// TwinCAT 3 PLC project Robotino_PLC_TEST
// ProgramVersion: 3.1.4022.0
// libraries:
//   Tc2_EtherCAT, * (Beckhoff Automation GmbH)
//   Tc2_Standard, * (Beckhoff Automation GmbH)
//   Tc2_System, * (Beckhoff Automation GmbH)
//   Tc2_Utilities, * (Beckhoff Automation GmbH)
//   Tc3_Module, * (Beckhoff Automation GmbH)
// project tree:
//   DUTs/ EnumState.TcDUT
//   / PlcTask.TcTTO
//   POUs/COE_Auswertung/ SDODaten.TcPOU, SDODatenMotor1.TcPOU, SDODatenMotor2.TcPOU, SDODatenMotor3.TcPOU, SDODatenMotorklemme1.TcPOU, SDODatenMotorklemme2.TcPOU
//   POUs/Motoransteuerung/ MAIN_Motoransteuerung.TcPOU
//   POUs/Motormesswerte/ MAIN_Motormesswerte.TcPOU
//   POUs/Shutdown/ MAIN_Shutdown.TcPOU, Shutdown.TcPOU
//   POUs/UDP/ MAIN_UDP.TcPOU, UDPConnect.TcPOU
// real-time tasks:
//   TASK PlcTask: cycle T#400us, priority 1, ADS port 350
//   TASK IrSensorTask: cycle T#1ms, priority 2, ADS port 351
//   TASK UdpTask: cycle T#2ms, priority 3, ADS port 352
//   TASK SimulinkTask: cycle T#5ms, priority 4, ADS port 353
// I/O:
//   DEVICE Gerät 1 (EtherCAT), AmsNetId 5.49.201.214.2.1
//     Klemme 1 (EK1200) [EK1200-5000 EtherCAT Netzteil (2A E-Bus)]
//       Motorklemme 1 [EL7342 2K. DC-Motor-Endstufe (50V, 3.5A)]
//       Motorklemme 2 [EL7342 2K. DC-Motor-Endstufe (50V, 3.5A)]
//       Digitale Eingänge [EL1008 8K. Dig. Eingang 24V, 3ms]
//       Digitale Ausgänge [EL2004 4K. Dig. Ausgang 24V, 0.5A]
//       Analoge Eingänge (8) [EL3068 8K. Ana. Eingang 0-10V]
//       Analog Eingänge (4) [EL3064 4K.Ana. Eingang 0-10V]
//       Netzklemme (5V) [EL9505 Netzteilklemme 5V]
//       Busendklemme [EL9011 Endklemme]
//   DEVICE UDP Adapter
// variable links:
//   Device 1 (EtherCAT) <-> irSensors/irSensors_Obj
//     Term 1 (EK1200)/Analog Eingänge (4)/AI Standard Channel 1/IR9 <-> Inputs/irInputData[8]
//     Term 1 (EK1200)/Analoge Eingänge (8)/AI Standard Channel {1..8}/IR{1..8} <-> Inputs/irInputData[{0..7}]  (8 links)
//   Robotino_PLC_TEST/Robotino_PLC_TEST Instance <-> Device 1 (EtherCAT)/Term 1 (EK1200)/Digitale Eingänge
//     PlcTask Inputs/MAIN_Motoransteuerung.bumper <-> Channel 2/Bumper
//     PlcTask Inputs/Shutdown.bStart <-> Channel 8/Shutdown
//   Robotino_PLC_TEST/Robotino_PLC_TEST Instance <-> Device 1 (EtherCAT)/Term 1 (EK1200)/Motorklemme 1
//     PlcTask Inputs/MAIN_Motormesswerte.encDataFromMotor2 <-> ENC Status compact Channel 2/Counter value
//     PlcTask Inputs/MAIN_Motormesswerte.encDataFromMotor3 <-> ENC Status compact Channel 1/Counter value
//     PlcTask Outputs/MAIN_Motoransteuerung.enableToMotor2 <-> DCM Control Channel 2/Control/Enable
//     PlcTask Outputs/MAIN_Motoransteuerung.enableToMotor3 <-> DCM Control Channel 1/Control/Enable
//     PlcTask Outputs/MAIN_Motoransteuerung.velocityToMotor2 <-> DCM Velocity Channel 2/Velocity
//     PlcTask Outputs/MAIN_Motoransteuerung.velocityToMotor3 <-> DCM Velocity Channel 1/Velocity
//   Robotino_PLC_TEST/Robotino_PLC_TEST Instance <-> Device 1 (EtherCAT)/Term 1 (EK1200)/Motorklemme 2
//     PlcTask Inputs/MAIN_Motormesswerte.encDataFromMotor1 <-> ENC Status compact Channel 1/Counter value
//     PlcTask Outputs/MAIN_Motoransteuerung.enableToMotor1 <-> DCM Control Channel 1/Control/Enable
//     PlcTask Outputs/MAIN_Motoransteuerung.velocityToMotor1 <-> DCM Velocity Channel 1/Velocity
//   Robotino_PLC_TEST/Robotino_PLC_TEST Instance <-> TcCOM Objects/Object2 (Gewerk3_Simulink_Regler)
//     PlcTask Inputs/MAIN_Motoransteuerung.vThetaCartesianToMotors <-> Output/thetaCartesianToMotors
//     PlcTask Inputs/MAIN_Motoransteuerung.vXCartesianToMotors <-> Output/vXCartesianToMotors
//     PlcTask Inputs/MAIN_Motoransteuerung.vYCartesianToMotors <-> Output/vYCartesianToMotors
//     PlcTask Outputs/MAIN_Motormesswerte.vXCartesianFromMotors <-> Input/u5elements[2]
//     PlcTask Outputs/MAIN_Motormesswerte.vYCartesianFromMotors <-> Input/u5elements[3]
//     PlcTask Outputs/MAIN_Motormesswerte.vthetaCartesianFromMotors <-> Input/u5elements[4]
//     PlcTask Outputs/MAIN_UDP.theta[4] <-> Input/UDP[11]
//     PlcTask Outputs/MAIN_UDP.x[4] <-> Input/UDP[9]
//     PlcTask Outputs/MAIN_UDP.y[4] <-> Input/UDP[10]

CONFIGURATION Robotino_PLC_TEST
    RESOURCE PLC ON TwinCAT3
        TASK PlcTask(INTERVAL := T#400us, PRIORITY := 1);
        PROGRAM MAIN_Motoransteuerung WITH PlcTask : MAIN_Motoransteuerung;
        PROGRAM MAIN_Motormesswerte WITH PlcTask : MAIN_Motormesswerte;
        PROGRAM MAIN_Shutdown WITH PlcTask : MAIN_Shutdown;
        PROGRAM MAIN_UDP WITH PlcTask : MAIN_UDP;
        PROGRAM SDODaten WITH PlcTask : SDODaten;
    END_RESOURCE
END_CONFIGURATION

// ---- DUTs/EnumState.TcDUT
{attribute 'qualified_only'}
{attribute 'strict'}
TYPE EnumState :
(
	init,
	drive,
	reset
);
END_TYPE

// ---- POUs/Motoransteuerung/MAIN_Motoransteuerung.TcPOU
PROGRAM MAIN_Motoransteuerung
VAR	
	//Zustandsautomat
	state:		EnumState:=EnumState.init;
	nextState:	EnumState:=EnumState.init;

	//Achsen Freischalten
	enableMotors: BOOL	:=0;

	//Umgerechnete Werte
	vX:		LREAL:=0;
	vY:		LREAL:=0;
	vTheta:	LREAL:=0;
	v1:		LREAL:=0;
	v2:		LREAL:=0;
	v3:		LREAL:=0;
	//Fahrrichtung Motor
	velocityMotor1 :LREAL:=0;
	velocityMotor2 :LREAL:=0;
	velocityMotor3 :LREAL:=0;
	
	//Skalierung auf MaxGeschwindigkeit Skalierung hängt mit CoE Register 8020:07 8020:08 zusammen !!!
	velocityMax:LREAL:=942.4777961;// Nenndrehzahl U/min CoE Register 8020:07 8020:08 fesgelegt Faktor 16 Wegen Getriebe 1:16
	velocityMotorsTf:LREAL:=0;
	
	// Skalierung auf Ansteuersignale LREAL=>WORD   Skalierung hängt mit CoE Register 8020:07 8020:08 zusammen !!!
	skalPos:LREAL:=34.7668668;//  MaxValue/MaxVelocity   [1/ mm/s]   32767/(942mm/s)   MaxVelocity=D*PI*n/(16*60) //16:1 Getriebeübersetzung  
	skalNeg:LREAL:=34.76792783;//  MaxVelau/MaxVelocity   [1/ mm/s]   32768/(942mm/s)   MaxVelocity=(80mm*PI*3600 U/min)/(16*60sec/min)
	
	//Inputs: CartesianToMotors + Bumper
	vXCartesianToMotors 	AT%I*:LREAL:=0;
	vYCartesianToMotors 	AT%I*:LREAL:=0;
	vThetaCartesianToMotors AT%I*:LREAL:=0;
	bumper	   AT%I*: BOOL:=0;
	
	//Outputs: Motor Values and Enable Signal
	enableToMotor1 AT%Q*:BOOL:=FALSE;
	enableToMotor2 AT%Q*:BOOL:=FALSE;
	enableToMotor3 AT%Q*:BOOL:=FALSE;
	
	velocityToMotor1 AT%Q*:INT:=0;
	velocityToMotor3 AT%Q*:INT:=0;
	velocityToMotor2 AT%Q*:INT:=0;
	
END_VAR

// Konverzierung ToMotors Anfang********************************************************

//	  conversion from positive and / or negative longitudinal, lateral and
//	  rotational velocities(in milimeters per second) to three separate
//	  positive motor velocities(resolution: 1Byte) and their rotation
//    direction
//inputs:  	velocityX  (longitudinal velocity in milimeters per second)
//         	velocityY  (lateral velocity in milimeters per second)
//			vtheta     (rotational velocity in milimeters per second)
//outputs : velocityToMotor1	
//			velocityToMotor2
//			velocityToMotor3
//conversion from longitudinal, lateral & rotational velocity to the
//three separate motor velocities
vX:=vXCartesianToMotors;
vY:=vYCartesianToMotors;
vTheta:=vThetaCartesianToMotors;

v1 := (-vX * COS(30.0*PI/180))	+ (vY * COS(60.0*PI/180))	+ (vTheta * 135.0);
v2 := 0.0						+ (-vY)						+ (vTheta * 135.0);
v3 := (vX * COS(30.0*PI/180))	+ (vY * COS(60.0*PI/180))	+ (vTheta * 135.0);
	
//Drehrichtung Umkehren
velocityMotor1:=-v1;
velocityMotor2:=-v2;
velocityMotor3:=-v3;

//Geschwindigkeitsbegrenzung
IF velocityMotor1 > velocityMax THEN
    velocityMotorsTf:= velocityMotor1;
    
    velocityMotor1:= velocityMax;
    velocityMotor2:= velocityMax * velocityMotor2 / velocityMotorsTf;
    velocityMotor3:= velocityMax * velocityMotor3 / velocityMotorsTf;
END_IF

IF velocityMotor2 > velocityMax THEN
    velocityMotorsTf:= velocityToMotor2;
    
    velocityMotor1:= velocityMax * velocityToMotor1 / velocityMotorsTf;
    velocityMotor2:= velocityMax;
    velocityMotor3:= velocityMax * velocityToMotor3 / velocityMotorsTf;
END_IF

IF velocityMotor3 > velocityMax THEN
    velocityMotorsTf:= velocityToMotor3;
    
    velocityMotor1:= velocityMax * velocityMotor1 / velocityMotorsTf;
    velocityMotor2:= velocityMax * velocityMotor2 / velocityMotorsTf;
    velocityMotor3:= velocityMax;
END_IF
// Konverzierung ToMotors ENDE********************************************************


//MOTORANSTEUERUNG Zustandsautomat

CASE state OF
	EnumState.init:						
						IF bumper=TRUE THEN
							nextState:=EnumState.reset;
							ELSE
								nextState:=EnumState.drive;
						END_IF
	EnumState.drive:
						IF velocityMotor1>=0 THEN
							velocityToMotor1:=LREAL_TO_INT(velocityMotor1*skalPos);
						ELSE
							velocityToMotor1:=LREAL_TO_INT(velocityMotor1*skalNeg);
						END_IF
						
						IF velocityMotor2>=0 THEN
							velocityToMotor2:=LREAL_TO_INT(velocityMotor2*skalPos);
						ELSE
							velocityToMotor2:=LREAL_TO_INT(velocityMotor2*skalNeg);
						END_IF
						
						IF velocityMotor3>=0 THEN
							velocityToMotor3:=LREAL_TO_INT(velocityMotor3*skalPos);
						ELSE
							velocityToMotor3:=LREAL_TO_INT(velocityMotor3*skalNeg); 
						END_IF
							
							enableToMotor1:=1;
							enableToMotor2:=1;
							enableToMotor3:=1;
							
						IF bumper=TRUE THEN
							nextState:=EnumState.reset;
						END_IF
	EnumState.reset:
						velocityToMotor1:=0;
						velocityToMotor2:=0;
						velocityToMotor3:=0;
						enableToMotor1:=0;
						enableToMotor2:=0;
						enableToMotor3:=0;
	ELSE
		nextState:=EnumState.reset;
END_CASE
state:=nextState;

END_PROGRAM

// ---- POUs/Motormesswerte/MAIN_Motormesswerte.TcPOU
PROGRAM MAIN_Motormesswerte
VAR
bStart: BOOL := FALSE;	

//ENC Daten Differenzieren für Geschwindigkeit
diffConst:LREAL:=0.0004;//SECONDS
encDataOldMotor1:UINT:=0;
encDataOldMotor2:UINT:=0;
encDataOldMotor3:UINT:=0;

//Koordinatentransformation Weg
skalEnc:LREAL:=0.00766990393;
x1:LREAL:=0;
x2:LREAL:=0;
x3:LREAL:=0;

xFromMotor1:LREAL:=0;
xFromMotor2:LREAL:=0;
xFromMotor3:LREAL:=0;

//Koordinatentransformation Geschwindigkeit
v1:LREAL:=0;
v2:LREAL:=0;
v3:LREAL:=0;
velocityFromMotor1:LREAL:=0;
velocityFromMotor2:LREAL:=0;
velocityFromMotor3:LREAL:=0;

//INPUTS
encDataFromMotor1 AT%I*  :UINT:=0;
encDataFromMotor2 AT%I*  :UINT:=0;
encDataFromMotor3 AT%I*  :UINT:=0;

diff:  INT :=0;
diff1: INT := 0;
diff2: INT := 0;
diff3: INT := 0;

//OUTPUTS
posXCartesianFromMotors AT%Q*:LREAL:=0;
posYCartesianFromMotors AT%Q*:LREAL:=0;
posThetaCartesianFromMotors AT%Q*:LREAL:=0;

vXCartesianFromMotors AT%Q*:LREAL:=0;
vYCartesianFromMotors AT%Q*:LREAL:=0;
vthetaCartesianFromMotors AT%Q*:LREAL:=0;
END_VAR

IF bStart = FALSE THEN
	encDataOldMotor1 := encDataFromMotor1;
	encDataOldMotor2 := encDataFromMotor2;
	encDataOldMotor3 := encDataFromMotor3;
	bStart := TRUE;
END_IF



// Encoder Wegberechnung und Differenzierung für Geschwindigkeit
diff1:=UINT_TO_INT(encDataFromMotor1) - UINT_TO_INT(encDataOldMotor1);
IF diff1 >= 32767 OR diff1 <= -32767 THEN
	diff1 := 0;
END_IF
diff2:=UINT_TO_INT(encDataFromMotor2) - UINT_TO_INT(encDataOldMotor2);
IF diff2 >= 32767 OR diff2 <= -32767 THEN
	diff2 := 0;
END_IF
diff3:=UINT_TO_INT(encDataFromMotor3) - UINT_TO_INT(encDataOldMotor3);
IF diff3 >= 32767 OR diff3 <= -32767 THEN
	diff3 := 0;
END_IF

xFromMotor1:=xFromMotor1+diff1*skalEnc;
velocityFromMotor1:=diff1/diffConst*skalEnc;

xFromMotor2:=xFromMotor2+diff2*skalEnc;
velocityFromMotor2:=diff2/diffConst*skalEnc;

xFromMotor3:=xFromMotor3+diff3*skalEnc;
velocityFromMotor3:=diff3/diffConst*skalEnc;

// Koordinatentransformation Weg
x1:=-xFromMotor1;
x2:=-xFromMotor2;
x3:=-xFromMotor3;

posXCartesianFromMotors:=(x3 - x1) / (2.0 * COS(30.0*PI/180));  //in mm / s
posYCartesianFromMotors:=(x1 - 2.0 * x2 + x3) / 3.0;            //in mm / s
posThetaCartesianFromMotors:=(x1 + x2 + x3) / (3.0 * 135.0);    //in rad / s

// Koordinatentransformation Geschwindigkeit
v1:=-velocityFromMotor1;
v2:=-velocityFromMotor2;
v3:=-velocityFromMotor3;

vXCartesianFromMotors:=(v3 - v1) / (2.0 * COS(30.0*PI/180));  //in mm / s
vYCartesianFromMotors:=(v1 - 2.0 * v2 + v3) / 3.0;            //in mm / s
vThetaCartesianFromMotors:=(v1 + v2 + v3) / (3.0 * 135.0);    //in rad / s

// Alte Encoderdaten speichern

encDataOldMotor1:=encDataFromMotor1;
encDataOldMotor2:=encDataFromMotor2;
encDataOldMotor3:=encDataFromMotor3;

END_PROGRAM

// ---- POUs/Shutdown/MAIN_Shutdown.TcPOU
PROGRAM MAIN_Shutdown
VAR
END_VAR

Shutdown();

END_PROGRAM

// ---- POUs/Shutdown/Shutdown.TcPOU
PROGRAM Shutdown
VAR
	bStart	AT%I* : BOOL := FALSE;
	Shutdown_Block: NT_Shutdown;
END_VAR

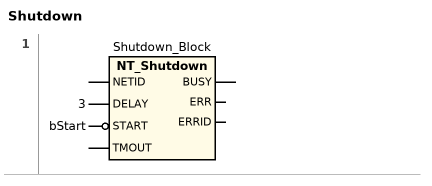
// NETWORK 1
Shutdown_Block(DELAY := 3, START := NOT bStart); // NT_Shutdown

END_PROGRAM

// ---- POUs/UDP/MAIN_UDP.TcPOU
PROGRAM MAIN_UDP
VAR
	//sPaketinhalt	: LREAL;
	//nPaketlaenge	: UDINT;
	
	x	  AT%Q*	: ARRAY[1..4] OF LREAL;
	y	  AT%Q*	: ARRAY[1..4] OF LREAL;
	theta AT%Q*	: ARRAY[1..4] OF LREAL;
	udp1 : UDPConnect;
END_VAR

udp1();

END_PROGRAM

// ---- POUs/UDP/UDPConnect.TcPOU
{attribute 'c++_compatible'}
FUNCTION_BLOCK UDPConnect IMPLEMENTS ITcIoUdpProtocolRecv
VAR_INPUT
END_VAR
VAR_OUTPUT
END_VAR
VAR
	{attribute 'TcInitSymbol'}
    oid:              OTCID; 
    ipUdp:            ITcIoUdpProtocol;
    updPort:          UINT := 25000;
    nReceivedPakets:  UINT;
    hrInit :          HRESULT;
    hrSend :          HRESULT;
END_VAR

IF ipUdp <> 0 THEN
    ipUdp.CheckReceived();
END_IF

METHOD FB_exit : BOOL
VAR_INPUT
	bInCopyCode : BOOL; // if TRUE, the exit method is called for exiting an instance that is copied afterwards (online change).
END_VAR
IF (NOT bInCopyCode AND ipUdp <> 0) THEN //Shutdown
     ipUdp.UnregisterReceiver(updPort);
    FW_SafeRelease(ADR(ipUdp));
     FB_exit := TRUE;
ELSE
     FB_exit := FALSE;
END_IF
END_METHOD

METHOD FB_init : BOOL
VAR_INPUT
	bInitRetains : BOOL; // if TRUE, the retain variables are initialized (warm start / cold start)
	bInCopyCode : BOOL;  // if TRUE, the instance afterwards gets moved into the copy code (online change)
END_VAR

VAR
    ipSrv: ITComObjectServer;
    hr : HRESULT;
END_VAR
IF NOT bInCopyCode THEN // no online change
    IF ipUdp = 0 THEN
     hrInit := FW_ObjMgr_GetObjectInstance(   oid:=oid, 
    
    iid:=TC_GLOBAL_IID_LIST.IID_ITcIoUdpProtocol, 

    pipUnk:=ADR(ipUdp) );
        IF ( SUCCEEDED(hr) AND ipUdp.RegisterReceiver(updPort, THIS^) = 0 ) THEN //open port
            FB_init := TRUE;
        ELSE
            FB_init := FALSE; 
            FW_SafeRelease(ADR(ipUdp));
        END_IF
    END_IF
END_IF
END_METHOD

METHOD FB_reinit : BOOL
VAR_INPUT
END_VAR
IF (ipUdp <> 0) THEN 
 ipUdp.RegisterReceiver(updPort, THIS^);
END_IF
END_METHOD

{attribute 'object_name' := 'ReceiveData'}
{attribute 'c++_compatible'}
{attribute 'signature_flag' := '33554688'}
{attribute 'pack_mode' := '4'}
{attribute 'show'}
{attribute 'minimal_input_size' := '4'}
METHOD ReceiveData : HRESULT
VAR_INPUT
	ipAddr	: UDINT;
	udpDestPort	: UINT;
	udpSrcPort	: UINT;
	nData	: UDINT;
	pData	: PVOID;
	pVlan	: POINTER TO ETYPE_VLAN_HEADER := 0;
END_VAR

VAR
	i	: ULINT := 0;
END_VAR
nReceivedPakets := nReceivedPakets+1;
//MAIN_UDP.nPaketlaenge := nData;

FOR i := 0 TO 3 DO
	memcpy(ADR(MAIN_UDP.x[i+1]),pData+((i*3)*8),8);
	memcpy(ADR(MAIN_UDP.y[i+1]),pData+((i*3+1)*8),8);
	memcpy(ADR(MAIN_UDP.theta[i+1]),pData+((i*3+2)*8),8);
END_FOR;
END_METHOD

{attribute 'c++_compatible'}
{attribute 'minimal_input_size' := '4'}
{attribute 'pack_mode' := '4'}
{warning 'Methodenimplementierung hinzufügen'}
METHOD TcAddRef : UDINT
END_METHOD

{attribute 'c++_compatible'}
{attribute 'minimal_input_size' := '4'}
{attribute 'pack_mode' := '4'}
{warning 'Methodenimplementierung hinzufügen'}
METHOD TcQueryInterface : HRESULT
VAR_INPUT
	iid	: REFERENCE TO IID;
	pipItf	: POINTER TO PVOID;
END_VAR
END_METHOD

{attribute 'c++_compatible'}
{attribute 'minimal_input_size' := '4'}
{attribute 'pack_mode' := '4'}
{warning 'Methodenimplementierung hinzufügen'}
METHOD TcRelease : UDINT
END_METHOD

END_FUNCTION_BLOCK

// ---- POUs/COE_Auswertung/SDODaten.TcPOU
PROGRAM SDODaten
VAR
	DatenMotor1: SDODatenMotor1;
	DatenMotor2: SDODatenMotor2;
	DatenMotor3: SDODatenMotor3;
	DatenMotorklemme1: SDODatenMotorklemme1;
	DatenMotorklemme2: SDODatenMotorklemme2;
END_VAR

DatenMotor1();
DatenMotor2();
DatenMotor3();
DatenMotorklemme1();
DatenMotorklemme2();

END_PROGRAM

// ---- POUs/COE_Auswertung/SDODatenMotor1.TcPOU
FUNCTION_BLOCK SDODatenMotor1
VAR_INPUT
END_VAR
VAR_OUTPUT
	
	Motor1Spannung: UINT;
	Motor1Strom: INT;
	Motor1Strombegrenzung: UINT;
	Motor1Regelfehler: INT;
	Motor1Geschwindigkeit: INT;
	Motor1Overloadtime: UINT;
	Motor1Overtemperature: BOOL;
	Motor1Torqueoverload: BOOL;
	Motor1Shortcirciut: BOOL;
	
END_VAR
VAR
	Motorspannung: FB_EcCoESdoRead;	
	Motorstrom: FB_EcCoESdoRead;
	Strombegrenzung: FB_EcCoESdoRead;
	Regelfehler: FB_EcCoESdoRead;
	Geschwindigkeit: FB_EcCoESdoRead;
	Overload: FB_EcCoESdoRead;
	Short_Circuit: FB_EcCoESdoRead;
	Torque_Overload: FB_EcCoESdoRead;
	Over_Temperature: FB_EcCoESdoRead;

	trigger: BOOL;
	TON_0: TON;
	TON_1: TON;
	ms: TIME;

END_VAR

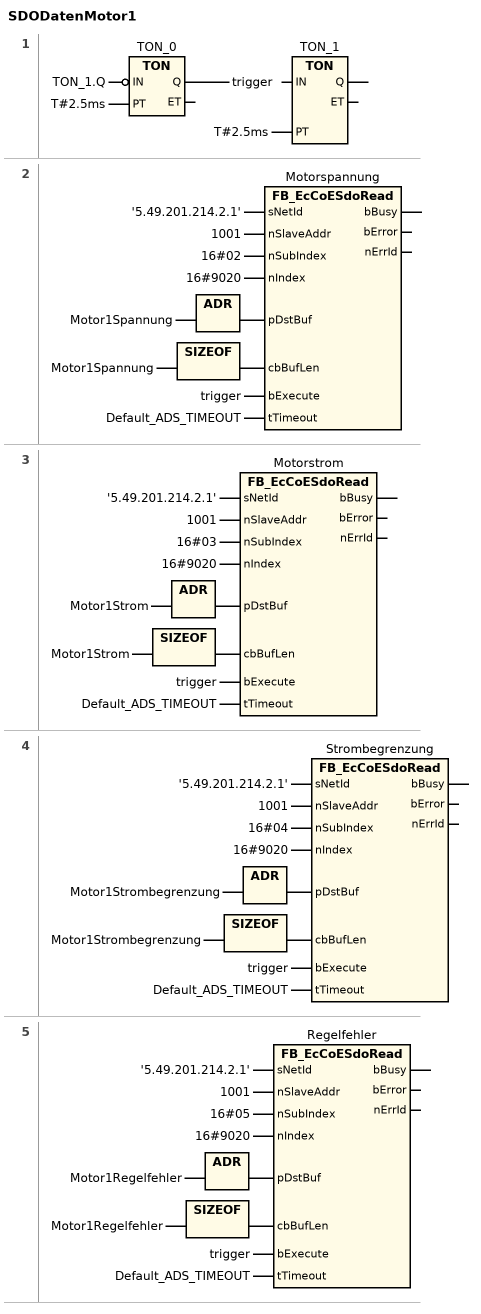
// NETWORK 1
TON_0(IN := NOT TON_1.Q, PT := T#2.5ms); // TON
trigger := TON_0.Q;
TON_1(IN := TON_0.Q, PT := T#2.5ms); // TON

// NETWORK 2
Motorspannung(
    sNetId := '5.49.201.214.2.1',
    nSlaveAddr := 1001,
    nSubIndex := 16#02,
    nIndex := 16#9020,
    pDstBuf := ADR(Motor1Spannung),
    cbBufLen := SIZEOF(Motor1Spannung),
    bExecute := trigger,
    tTimeout := Default_ADS_TIMEOUT); // FB_EcCoESdoRead

// NETWORK 3
Motorstrom(
    sNetId := '5.49.201.214.2.1',
    nSlaveAddr := 1001,
    nSubIndex := 16#03,
    nIndex := 16#9020,
    pDstBuf := ADR(Motor1Strom),
    cbBufLen := SIZEOF(Motor1Strom),
    bExecute := trigger,
    tTimeout := Default_ADS_TIMEOUT); // FB_EcCoESdoRead

// NETWORK 4
Strombegrenzung(
    sNetId := '5.49.201.214.2.1',
    nSlaveAddr := 1001,
    nSubIndex := 16#04,
    nIndex := 16#9020,
    pDstBuf := ADR(Motor1Strombegrenzung),
    cbBufLen := SIZEOF(Motor1Strombegrenzung),
    bExecute := trigger,
    tTimeout := Default_ADS_TIMEOUT); // FB_EcCoESdoRead

// NETWORK 5
Regelfehler(
    sNetId := '5.49.201.214.2.1',
    nSlaveAddr := 1001,
    nSubIndex := 16#05,
    nIndex := 16#9020,
    pDstBuf := ADR(Motor1Regelfehler),
    cbBufLen := SIZEOF(Motor1Regelfehler),
    bExecute := trigger,
    tTimeout := Default_ADS_TIMEOUT); // FB_EcCoESdoRead

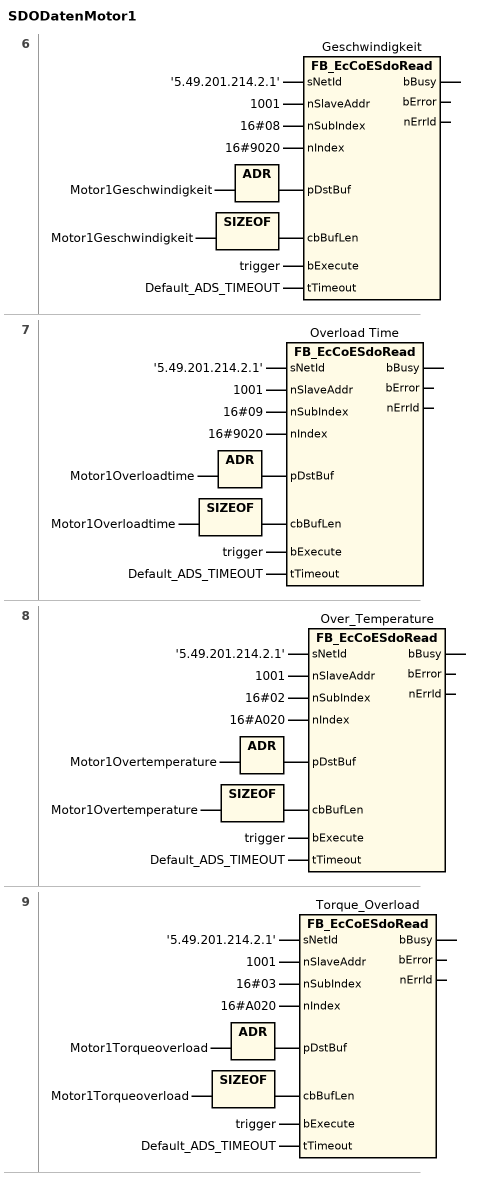
// NETWORK 6
Geschwindigkeit(
    sNetId := '5.49.201.214.2.1',
    nSlaveAddr := 1001,
    nSubIndex := 16#08,
    nIndex := 16#9020,
    pDstBuf := ADR(Motor1Geschwindigkeit),
    cbBufLen := SIZEOF(Motor1Geschwindigkeit),
    bExecute := trigger,
    tTimeout := Default_ADS_TIMEOUT); // FB_EcCoESdoRead

// NETWORK 7
Overload Time(
    sNetId := '5.49.201.214.2.1',
    nSlaveAddr := 1001,
    nSubIndex := 16#09,
    nIndex := 16#9020,
    pDstBuf := ADR(Motor1Overloadtime),
    cbBufLen := SIZEOF(Motor1Overloadtime),
    bExecute := trigger,
    tTimeout := Default_ADS_TIMEOUT); // FB_EcCoESdoRead

// NETWORK 8
Over_Temperature(
    sNetId := '5.49.201.214.2.1',
    nSlaveAddr := 1001,
    nSubIndex := 16#02,
    nIndex := 16#A020,
    pDstBuf := ADR(Motor1Overtemperature),
    cbBufLen := SIZEOF(Motor1Overtemperature),
    bExecute := trigger,
    tTimeout := Default_ADS_TIMEOUT); // FB_EcCoESdoRead

// NETWORK 9
Torque_Overload(
    sNetId := '5.49.201.214.2.1',
    nSlaveAddr := 1001,
    nSubIndex := 16#03,
    nIndex := 16#A020,
    pDstBuf := ADR(Motor1Torqueoverload),
    cbBufLen := SIZEOF(Motor1Torqueoverload),
    bExecute := trigger,
    tTimeout := Default_ADS_TIMEOUT); // FB_EcCoESdoRead

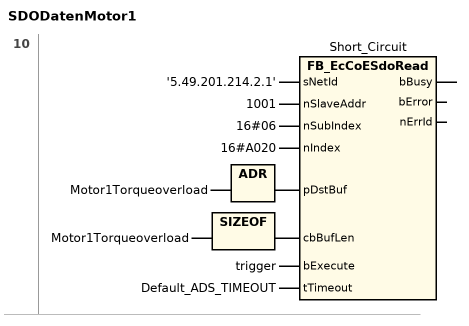
// NETWORK 10
Short_Circuit(
    sNetId := '5.49.201.214.2.1',
    nSlaveAddr := 1001,
    nSubIndex := 16#06,
    nIndex := 16#A020,
    pDstBuf := ADR(Motor1Torqueoverload),
    cbBufLen := SIZEOF(Motor1Torqueoverload),
    bExecute := trigger,
    tTimeout := Default_ADS_TIMEOUT); // FB_EcCoESdoRead

END_FUNCTION_BLOCK

// ---- POUs/COE_Auswertung/SDODatenMotor2.TcPOU
FUNCTION_BLOCK SDODatenMotor2
VAR_INPUT
END_VAR
VAR_OUTPUT
	
	Motor2Spannung: UINT;
	Motor2Strom: INT;
	Motor2Strombegrenzung: UINT;
	Motor2Regelfehler: INT;
	Motor2Geschwindigkeit: INT;
	Motor2Overloadtime: UINT;
	Motor2Overtemperature: BOOL;
	Motor2Torqueoverload: BOOL;
	Motor2Shortcirciut: BOOL;
	
END_VAR
VAR
	Motorspannung: FB_EcCoESdoRead;	
	Motorstrom: FB_EcCoESdoRead;
	Strombegrenzung: FB_EcCoESdoRead;
	Regelfehler: FB_EcCoESdoRead;
	Geschwindigkeit: FB_EcCoESdoRead;
	Overload: FB_EcCoESdoRead;
	Short_Circuit: FB_EcCoESdoRead;
	Torque_Overload: FB_EcCoESdoRead;
	Over_Temperature: FB_EcCoESdoRead;

	trigger: BOOL;
	TON_0: TON;
	TON_1: TON;
	ms: TIME;

END_VAR

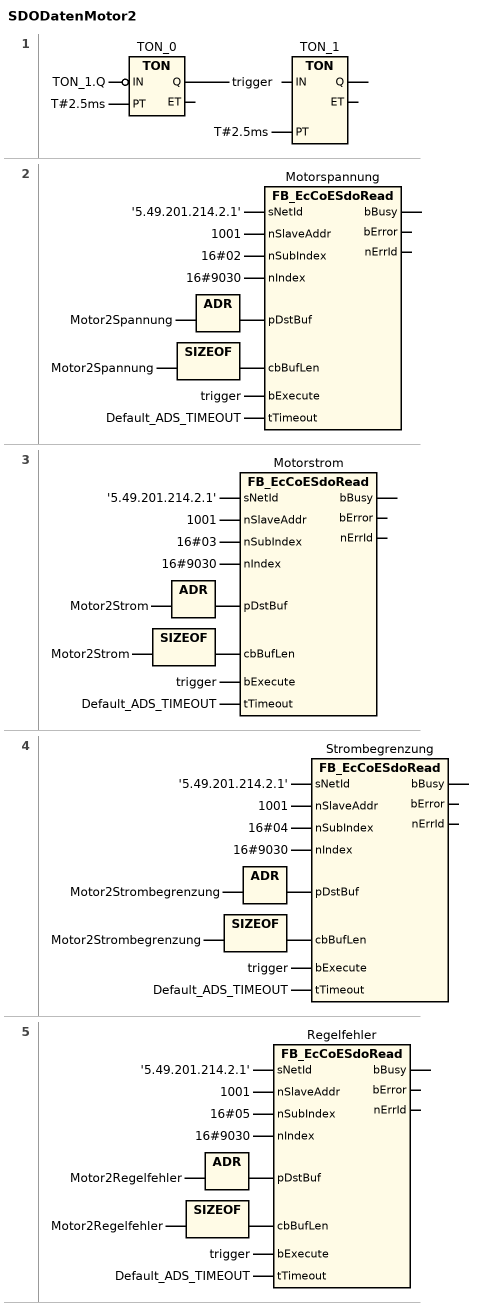
// NETWORK 1
TON_0(IN := NOT TON_1.Q, PT := T#2.5ms); // TON
trigger := TON_0.Q;
TON_1(IN := TON_0.Q, PT := T#2.5ms); // TON

// NETWORK 2
Motorspannung(
    sNetId := '5.49.201.214.2.1',
    nSlaveAddr := 1001,
    nSubIndex := 16#02,
    nIndex := 16#9030,
    pDstBuf := ADR(Motor2Spannung),
    cbBufLen := SIZEOF(Motor2Spannung),
    bExecute := trigger,
    tTimeout := Default_ADS_TIMEOUT); // FB_EcCoESdoRead

// NETWORK 3
Motorstrom(
    sNetId := '5.49.201.214.2.1',
    nSlaveAddr := 1001,
    nSubIndex := 16#03,
    nIndex := 16#9030,
    pDstBuf := ADR(Motor2Strom),
    cbBufLen := SIZEOF(Motor2Strom),
    bExecute := trigger,
    tTimeout := Default_ADS_TIMEOUT); // FB_EcCoESdoRead

// NETWORK 4
Strombegrenzung(
    sNetId := '5.49.201.214.2.1',
    nSlaveAddr := 1001,
    nSubIndex := 16#04,
    nIndex := 16#9030,
    pDstBuf := ADR(Motor2Strombegrenzung),
    cbBufLen := SIZEOF(Motor2Strombegrenzung),
    bExecute := trigger,
    tTimeout := Default_ADS_TIMEOUT); // FB_EcCoESdoRead

// NETWORK 5
Regelfehler(
    sNetId := '5.49.201.214.2.1',
    nSlaveAddr := 1001,
    nSubIndex := 16#05,
    nIndex := 16#9030,
    pDstBuf := ADR(Motor2Regelfehler),
    cbBufLen := SIZEOF(Motor2Regelfehler),
    bExecute := trigger,
    tTimeout := Default_ADS_TIMEOUT); // FB_EcCoESdoRead

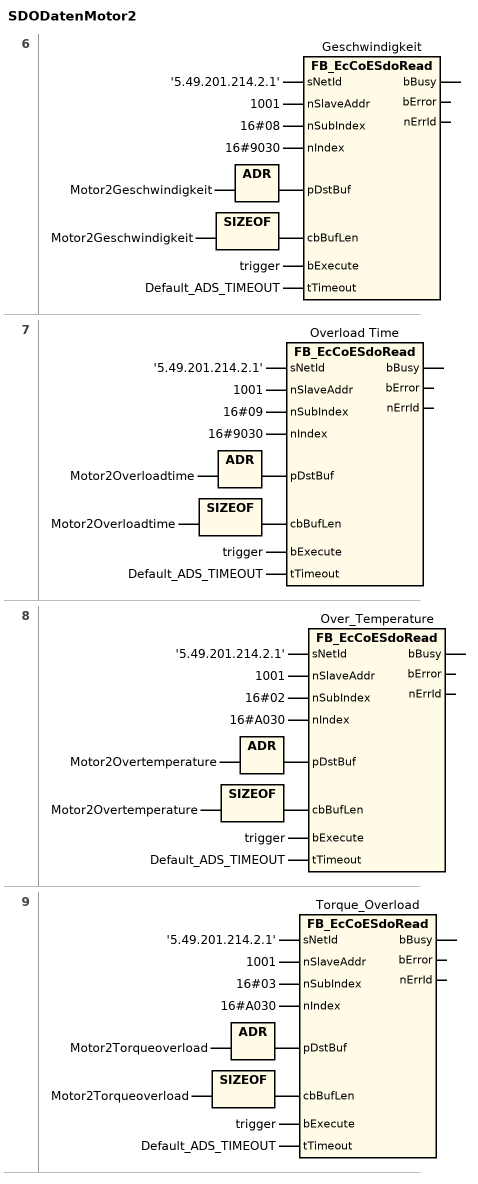
// NETWORK 6
Geschwindigkeit(
    sNetId := '5.49.201.214.2.1',
    nSlaveAddr := 1001,
    nSubIndex := 16#08,
    nIndex := 16#9030,
    pDstBuf := ADR(Motor2Geschwindigkeit),
    cbBufLen := SIZEOF(Motor2Geschwindigkeit),
    bExecute := trigger,
    tTimeout := Default_ADS_TIMEOUT); // FB_EcCoESdoRead

// NETWORK 7
Overload Time(
    sNetId := '5.49.201.214.2.1',
    nSlaveAddr := 1001,
    nSubIndex := 16#09,
    nIndex := 16#9030,
    pDstBuf := ADR(Motor2Overloadtime),
    cbBufLen := SIZEOF(Motor2Overloadtime),
    bExecute := trigger,
    tTimeout := Default_ADS_TIMEOUT); // FB_EcCoESdoRead

// NETWORK 8
Over_Temperature(
    sNetId := '5.49.201.214.2.1',
    nSlaveAddr := 1001,
    nSubIndex := 16#02,
    nIndex := 16#A030,
    pDstBuf := ADR(Motor2Overtemperature),
    cbBufLen := SIZEOF(Motor2Overtemperature),
    bExecute := trigger,
    tTimeout := Default_ADS_TIMEOUT); // FB_EcCoESdoRead

// NETWORK 9
Torque_Overload(
    sNetId := '5.49.201.214.2.1',
    nSlaveAddr := 1001,
    nSubIndex := 16#03,
    nIndex := 16#A030,
    pDstBuf := ADR(Motor2Torqueoverload),
    cbBufLen := SIZEOF(Motor2Torqueoverload),
    bExecute := trigger,
    tTimeout := Default_ADS_TIMEOUT); // FB_EcCoESdoRead

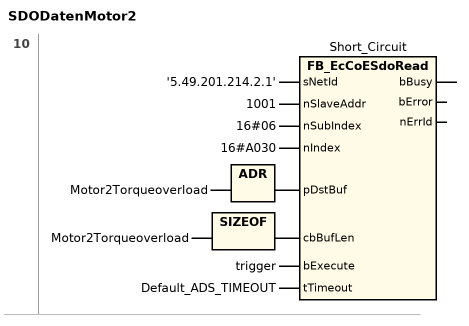
// NETWORK 10
Short_Circuit(
    sNetId := '5.49.201.214.2.1',
    nSlaveAddr := 1001,
    nSubIndex := 16#06,
    nIndex := 16#A030,
    pDstBuf := ADR(Motor2Torqueoverload),
    cbBufLen := SIZEOF(Motor2Torqueoverload),
    bExecute := trigger,
    tTimeout := Default_ADS_TIMEOUT); // FB_EcCoESdoRead

END_FUNCTION_BLOCK

// ---- POUs/COE_Auswertung/SDODatenMotor3.TcPOU
FUNCTION_BLOCK SDODatenMotor3
VAR_INPUT
END_VAR
VAR_OUTPUT
	
	Motor3Spannung: UINT;
	Motor3Strom: INT;
	Motor3Strombegrenzung: UINT;
	Motor3Regelfehler: INT;
	Motor3Geschwindigkeit: INT;
	Motor3Overloadtime: UINT;
	Motor3Overtemperature: BOOL;
	Motor3Torqueoverload: BOOL;
	Motor3Shortcirciut: BOOL;
	
END_VAR
VAR
	Motorspannung: FB_EcCoESdoRead;	
	Motorstrom: FB_EcCoESdoRead;
	Strombegrenzung: FB_EcCoESdoRead;
	Regelfehler: FB_EcCoESdoRead;
	Geschwindigkeit: FB_EcCoESdoRead;
	Overload: FB_EcCoESdoRead;
	Short_Circuit: FB_EcCoESdoRead;
	Torque_Overload: FB_EcCoESdoRead;
	Over_Temperature: FB_EcCoESdoRead;

	trigger: BOOL;
	TON_0: TON;
	TON_1: TON;
	ms: TIME;

END_VAR

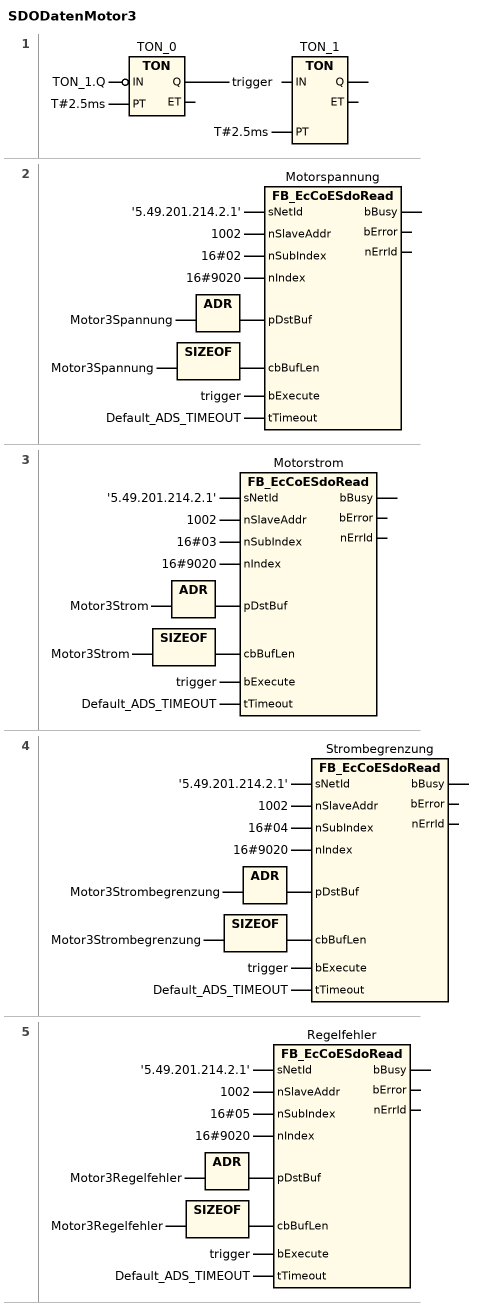
// NETWORK 1
TON_0(IN := NOT TON_1.Q, PT := T#2.5ms); // TON
trigger := TON_0.Q;
TON_1(IN := TON_0.Q, PT := T#2.5ms); // TON

// NETWORK 2
Motorspannung(
    sNetId := '5.49.201.214.2.1',
    nSlaveAddr := 1002,
    nSubIndex := 16#02,
    nIndex := 16#9020,
    pDstBuf := ADR(Motor3Spannung),
    cbBufLen := SIZEOF(Motor3Spannung),
    bExecute := trigger,
    tTimeout := Default_ADS_TIMEOUT); // FB_EcCoESdoRead

// NETWORK 3
Motorstrom(
    sNetId := '5.49.201.214.2.1',
    nSlaveAddr := 1002,
    nSubIndex := 16#03,
    nIndex := 16#9020,
    pDstBuf := ADR(Motor3Strom),
    cbBufLen := SIZEOF(Motor3Strom),
    bExecute := trigger,
    tTimeout := Default_ADS_TIMEOUT); // FB_EcCoESdoRead

// NETWORK 4
Strombegrenzung(
    sNetId := '5.49.201.214.2.1',
    nSlaveAddr := 1002,
    nSubIndex := 16#04,
    nIndex := 16#9020,
    pDstBuf := ADR(Motor3Strombegrenzung),
    cbBufLen := SIZEOF(Motor3Strombegrenzung),
    bExecute := trigger,
    tTimeout := Default_ADS_TIMEOUT); // FB_EcCoESdoRead

// NETWORK 5
Regelfehler(
    sNetId := '5.49.201.214.2.1',
    nSlaveAddr := 1002,
    nSubIndex := 16#05,
    nIndex := 16#9020,
    pDstBuf := ADR(Motor3Regelfehler),
    cbBufLen := SIZEOF(Motor3Regelfehler),
    bExecute := trigger,
    tTimeout := Default_ADS_TIMEOUT); // FB_EcCoESdoRead

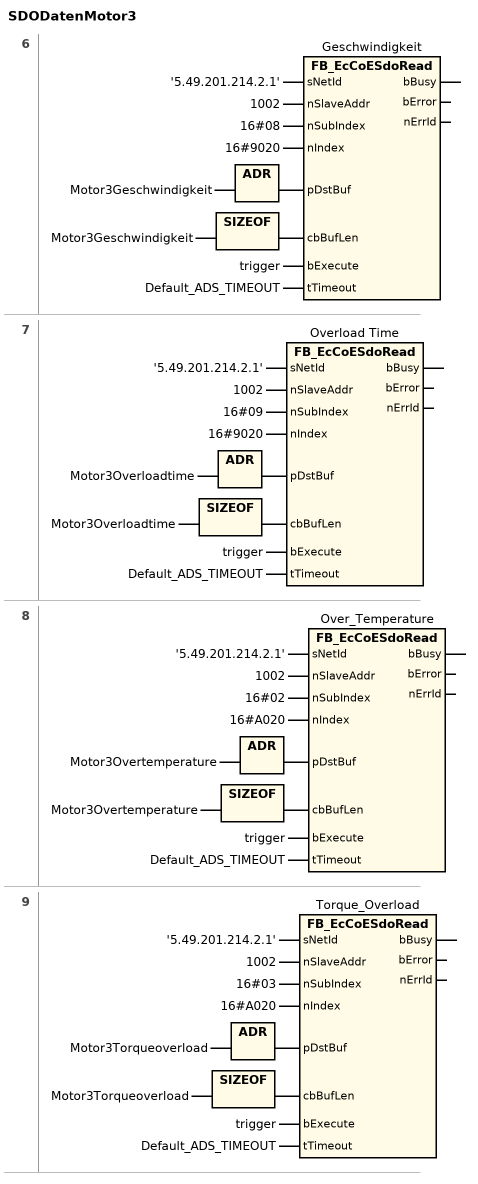
// NETWORK 6
Geschwindigkeit(
    sNetId := '5.49.201.214.2.1',
    nSlaveAddr := 1002,
    nSubIndex := 16#08,
    nIndex := 16#9020,
    pDstBuf := ADR(Motor3Geschwindigkeit),
    cbBufLen := SIZEOF(Motor3Geschwindigkeit),
    bExecute := trigger,
    tTimeout := Default_ADS_TIMEOUT); // FB_EcCoESdoRead

// NETWORK 7
Overload Time(
    sNetId := '5.49.201.214.2.1',
    nSlaveAddr := 1002,
    nSubIndex := 16#09,
    nIndex := 16#9020,
    pDstBuf := ADR(Motor3Overloadtime),
    cbBufLen := SIZEOF(Motor3Overloadtime),
    bExecute := trigger,
    tTimeout := Default_ADS_TIMEOUT); // FB_EcCoESdoRead

// NETWORK 8
Over_Temperature(
    sNetId := '5.49.201.214.2.1',
    nSlaveAddr := 1002,
    nSubIndex := 16#02,
    nIndex := 16#A020,
    pDstBuf := ADR(Motor3Overtemperature),
    cbBufLen := SIZEOF(Motor3Overtemperature),
    bExecute := trigger,
    tTimeout := Default_ADS_TIMEOUT); // FB_EcCoESdoRead

// NETWORK 9
Torque_Overload(
    sNetId := '5.49.201.214.2.1',
    nSlaveAddr := 1002,
    nSubIndex := 16#03,
    nIndex := 16#A020,
    pDstBuf := ADR(Motor3Torqueoverload),
    cbBufLen := SIZEOF(Motor3Torqueoverload),
    bExecute := trigger,
    tTimeout := Default_ADS_TIMEOUT); // FB_EcCoESdoRead

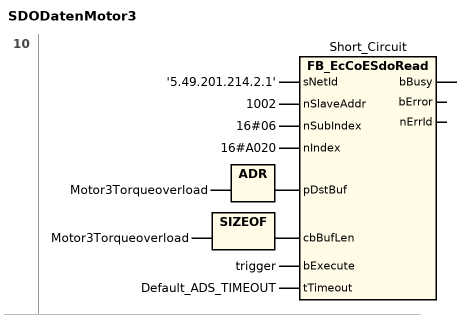
// NETWORK 10
Short_Circuit(
    sNetId := '5.49.201.214.2.1',
    nSlaveAddr := 1002,
    nSubIndex := 16#06,
    nIndex := 16#A020,
    pDstBuf := ADR(Motor3Torqueoverload),
    cbBufLen := SIZEOF(Motor3Torqueoverload),
    bExecute := trigger,
    tTimeout := Default_ADS_TIMEOUT); // FB_EcCoESdoRead

END_FUNCTION_BLOCK

// ---- POUs/COE_Auswertung/SDODatenMotorklemme1.TcPOU
FUNCTION_BLOCK SDODatenMotorklemme1
VAR_INPUT
END_VAR
VAR_OUTPUT
	
	Motorklemme1Internaltemperature: SINT;
	Motorklemme1Steuerspannung: UINT;
	Motorklemme1Lastspannung: UINT;
	Motorklemme1Zykluszeit: UINT;
	Motorklemme1PWMFrequency: UINT;
		
END_VAR
VAR

	Internal_Temperature: FB_EcCoESdoRead;
	Control_Voltage: FB_EcCoESdoRead;
	Supply_Voltage: FB_EcCoESdoRead;
	Cycletime: FB_EcCoESdoRead;
	PWM_Frequency: FB_EcCoESdoRead;
	
	trigger: BOOL;
	TON_0: TON;
	TON_1: TON;
	ms: TIME;

END_VAR

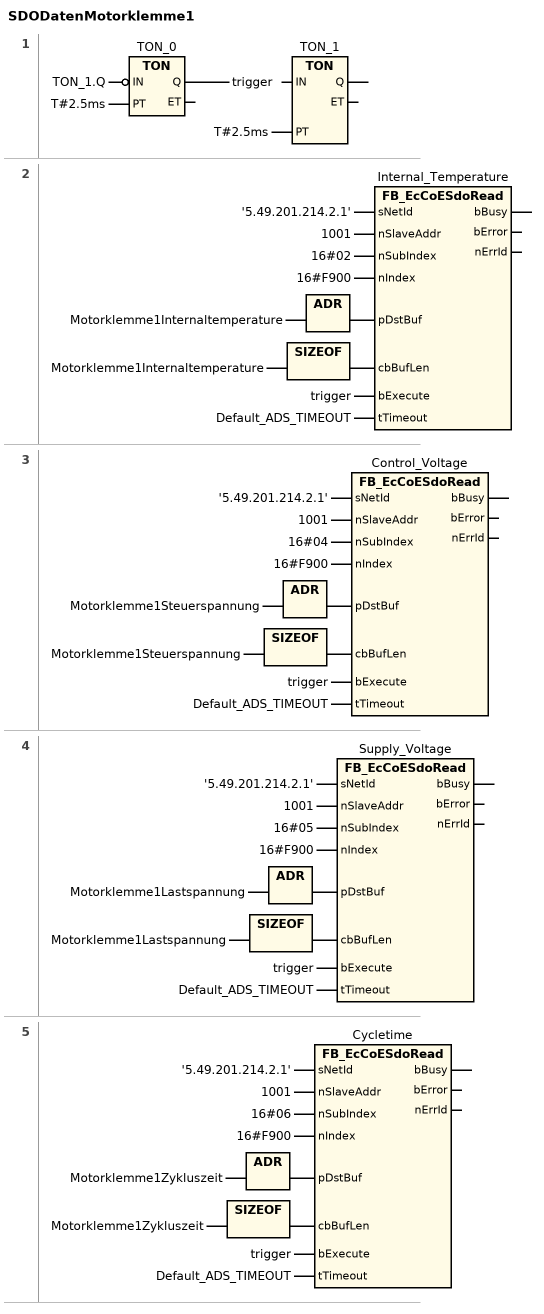
// NETWORK 1
TON_0(IN := NOT TON_1.Q, PT := T#2.5ms); // TON
trigger := TON_0.Q;
TON_1(IN := TON_0.Q, PT := T#2.5ms); // TON

// NETWORK 2
Internal_Temperature(
    sNetId := '5.49.201.214.2.1',
    nSlaveAddr := 1001,
    nSubIndex := 16#02,
    nIndex := 16#F900,
    pDstBuf := ADR(Motorklemme1Internaltemperature),
    cbBufLen := SIZEOF(Motorklemme1Internaltemperature),
    bExecute := trigger,
    tTimeout := Default_ADS_TIMEOUT); // FB_EcCoESdoRead

// NETWORK 3
Control_Voltage(
    sNetId := '5.49.201.214.2.1',
    nSlaveAddr := 1001,
    nSubIndex := 16#04,
    nIndex := 16#F900,
    pDstBuf := ADR(Motorklemme1Steuerspannung),
    cbBufLen := SIZEOF(Motorklemme1Steuerspannung),
    bExecute := trigger,
    tTimeout := Default_ADS_TIMEOUT); // FB_EcCoESdoRead

// NETWORK 4
Supply_Voltage(
    sNetId := '5.49.201.214.2.1',
    nSlaveAddr := 1001,
    nSubIndex := 16#05,
    nIndex := 16#F900,
    pDstBuf := ADR(Motorklemme1Lastspannung),
    cbBufLen := SIZEOF(Motorklemme1Lastspannung),
    bExecute := trigger,
    tTimeout := Default_ADS_TIMEOUT); // FB_EcCoESdoRead

// NETWORK 5
Cycletime(
    sNetId := '5.49.201.214.2.1',
    nSlaveAddr := 1001,
    nSubIndex := 16#06,
    nIndex := 16#F900,
    pDstBuf := ADR(Motorklemme1Zykluszeit),
    cbBufLen := SIZEOF(Motorklemme1Zykluszeit),
    bExecute := trigger,
    tTimeout := Default_ADS_TIMEOUT); // FB_EcCoESdoRead

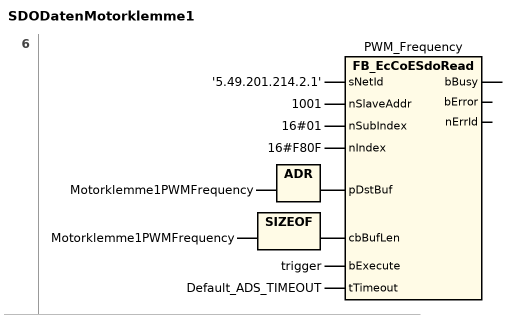
// NETWORK 6
PWM_Frequency(
    sNetId := '5.49.201.214.2.1',
    nSlaveAddr := 1001,
    nSubIndex := 16#01,
    nIndex := 16#F80F,
    pDstBuf := ADR(Motorklemme1PWMFrequency),
    cbBufLen := SIZEOF(Motorklemme1PWMFrequency),
    bExecute := trigger,
    tTimeout := Default_ADS_TIMEOUT); // FB_EcCoESdoRead

END_FUNCTION_BLOCK

// ---- POUs/COE_Auswertung/SDODatenMotorklemme2.TcPOU
FUNCTION_BLOCK SDODatenMotorklemme2
VAR_INPUT
END_VAR
VAR_OUTPUT
	
	Motorklemme1Internaltemperature: SINT;
	Motorklemme1Steuerspannung: UINT;
	Motorklemme1Lastspannung: UINT;
	Motorklemme1Zykluszeit: UINT;
	Motorklemme1PWMFrequency: UINT;
		
END_VAR
VAR

	Internal_Temperature: FB_EcCoESdoRead;
	Control_Voltage: FB_EcCoESdoRead;
	Supply_Voltage: FB_EcCoESdoRead;
	Cycletime: FB_EcCoESdoRead;
	PWM_Frequency: FB_EcCoESdoRead;
	
	trigger: BOOL;
	TON_0: TON;
	TON_1: TON;
	ms: TIME;

END_VAR

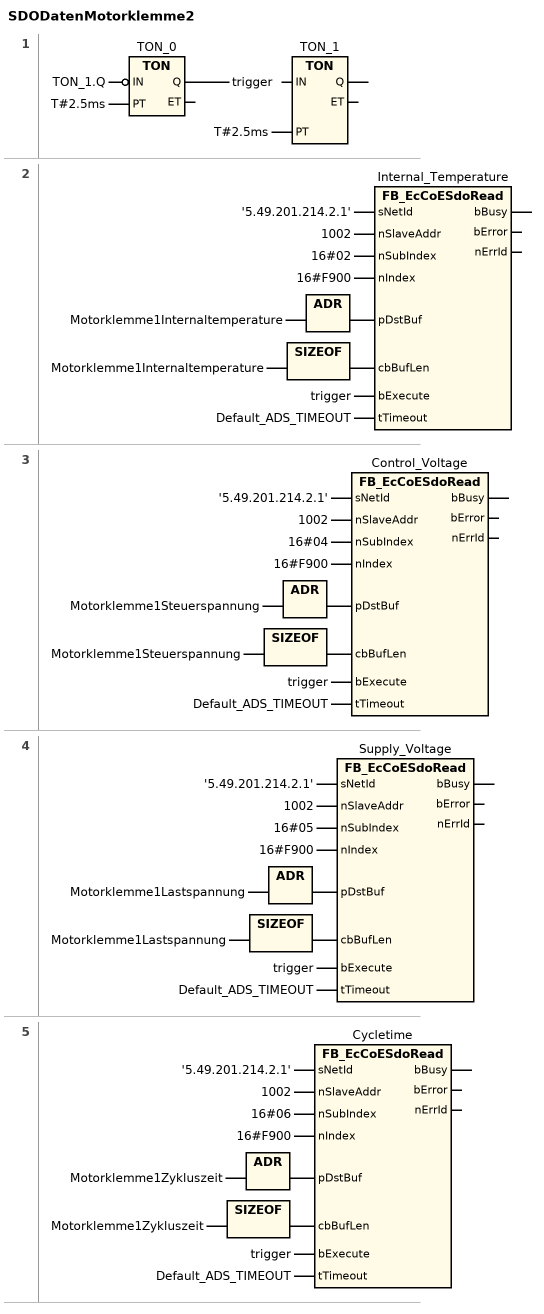
// NETWORK 1
TON_0(IN := NOT TON_1.Q, PT := T#2.5ms); // TON
trigger := TON_0.Q;
TON_1(IN := TON_0.Q, PT := T#2.5ms); // TON

// NETWORK 2
Internal_Temperature(
    sNetId := '5.49.201.214.2.1',
    nSlaveAddr := 1002,
    nSubIndex := 16#02,
    nIndex := 16#F900,
    pDstBuf := ADR(Motorklemme1Internaltemperature),
    cbBufLen := SIZEOF(Motorklemme1Internaltemperature),
    bExecute := trigger,
    tTimeout := Default_ADS_TIMEOUT); // FB_EcCoESdoRead

// NETWORK 3
Control_Voltage(
    sNetId := '5.49.201.214.2.1',
    nSlaveAddr := 1002,
    nSubIndex := 16#04,
    nIndex := 16#F900,
    pDstBuf := ADR(Motorklemme1Steuerspannung),
    cbBufLen := SIZEOF(Motorklemme1Steuerspannung),
    bExecute := trigger,
    tTimeout := Default_ADS_TIMEOUT); // FB_EcCoESdoRead

// NETWORK 4
Supply_Voltage(
    sNetId := '5.49.201.214.2.1',
    nSlaveAddr := 1002,
    nSubIndex := 16#05,
    nIndex := 16#F900,
    pDstBuf := ADR(Motorklemme1Lastspannung),
    cbBufLen := SIZEOF(Motorklemme1Lastspannung),
    bExecute := trigger,
    tTimeout := Default_ADS_TIMEOUT); // FB_EcCoESdoRead

// NETWORK 5
Cycletime(
    sNetId := '5.49.201.214.2.1',
    nSlaveAddr := 1002,
    nSubIndex := 16#06,
    nIndex := 16#F900,
    pDstBuf := ADR(Motorklemme1Zykluszeit),
    cbBufLen := SIZEOF(Motorklemme1Zykluszeit),
    bExecute := trigger,
    tTimeout := Default_ADS_TIMEOUT); // FB_EcCoESdoRead

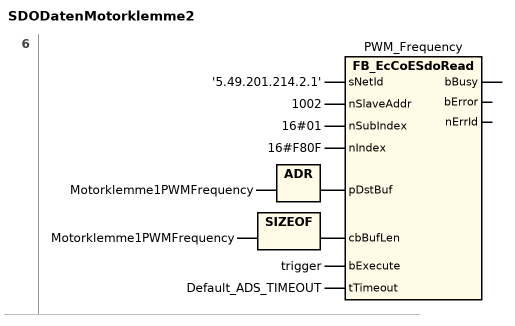
// NETWORK 6
PWM_Frequency(
    sNetId := '5.49.201.214.2.1',
    nSlaveAddr := 1002,
    nSubIndex := 16#01,
    nIndex := 16#F80F,
    pDstBuf := ADR(Motorklemme1PWMFrequency),
    cbBufLen := SIZEOF(Motorklemme1PWMFrequency),
    bExecute := trigger,
    tTimeout := Default_ADS_TIMEOUT); // FB_EcCoESdoRead

END_FUNCTION_BLOCK
